Fanuc KAREL source: V_ACQ_VAMAP.kl

PROGRAM T
%NOLOCKGROUP
VAR
 v0 : STRING[40]
 v1 : BOOLEAN
 v2 : VECTOR
 v3 : INTEGER
BEGIN
 V_ACQ_VAMAP(v0, v1, v2, v3)
END T
